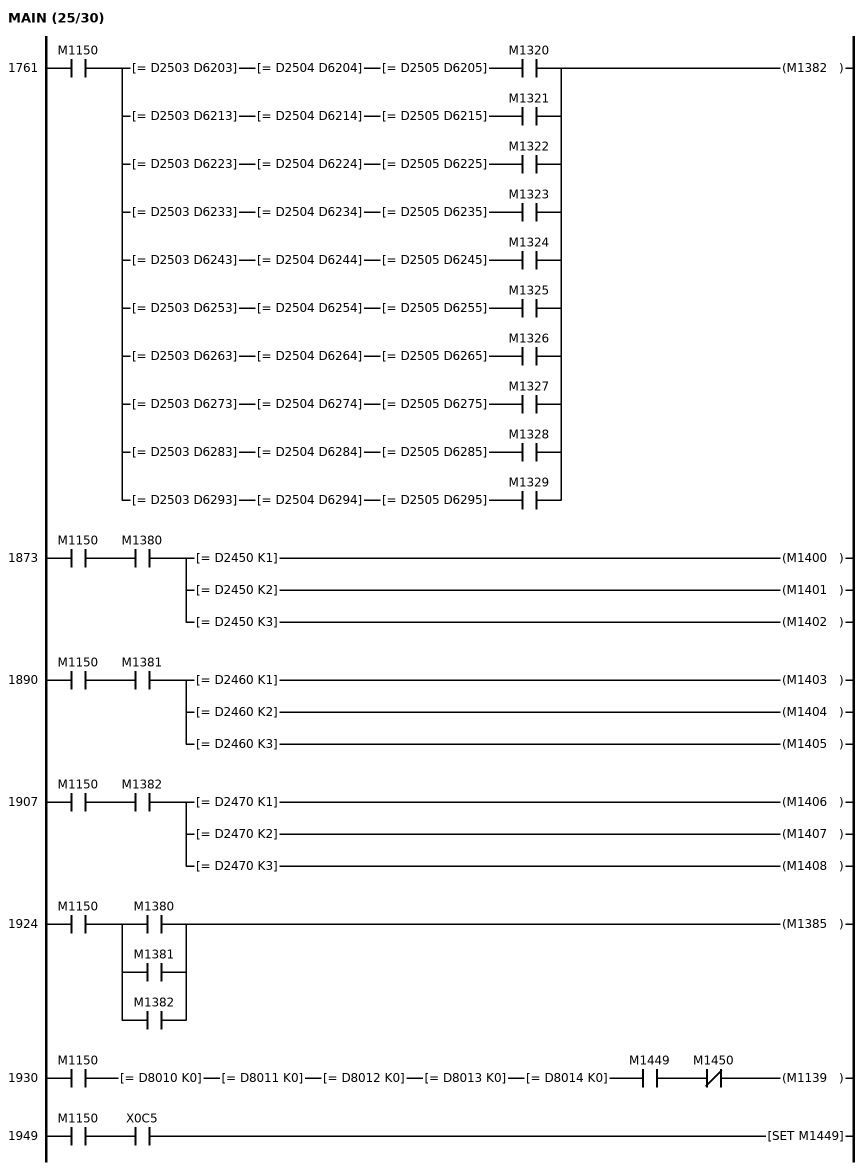
[picture p24: ladder of MAIN, rungs at steps 1761 to 1949]
1761  LD      M1150
      LD=     D2503 D6203
      AND=    D2504 D6204
      AND=    D2505 D6205
      AND     M1320
      LD=     D2503 D6213
      AND=    D2504 D6214
      AND=    D2505 D6215
      AND     M1321
      ORB
      LD=     D2503 D6223
      AND=    D2504 D6224
      AND=    D2505 D6225
      AND     M1322
      ORB
      LD=     D2503 D6233
      AND=    D2504 D6234
      AND=    D2505 D6235
      AND     M1323
      ORB
      LD=     D2503 D6243
      AND=    D2504 D6244
      AND=    D2505 D6245
      AND     M1324
      ORB
      LD=     D2503 D6253
      AND=    D2504 D6254
      AND=    D2505 D6255
      AND     M1325
      ORB
      LD=     D2503 D6263
      AND=    D2504 D6264
      AND=    D2505 D6265
      AND     M1326
      ORB
      LD=     D2503 D6273
      AND=    D2504 D6274
      AND=    D2505 D6275
      AND     M1327
      ORB
      LD=     D2503 D6283
      AND=    D2504 D6284
      AND=    D2505 D6285
      AND     M1328
      ORB
      LD=     D2503 D6293
      AND=    D2504 D6294
      AND=    D2505 D6295
      AND     M1329
      ORB
      ANB
      OUT     M1382
1873  LD      M1150
      AND     M1380
      MPS
      AND=    D2450 K1
      OUT     M1400
      MRD
      AND=    D2450 K2
      OUT     M1401
      MPP
      AND=    D2450 K3
      OUT     M1402
1890  LD      M1150
      AND     M1381
      MPS
      AND=    D2460 K1
      OUT     M1403
      MRD
      AND=    D2460 K2
      OUT     M1404
      MPP
      AND=    D2460 K3
      OUT     M1405
1907  LD      M1150
      AND     M1382
      MPS
      AND=    D2470 K1
      OUT     M1406
      MRD
      AND=    D2470 K2
      OUT     M1407
      MPP
      AND=    D2470 K3
      OUT     M1408
1924  LD      M1150
      LD      M1380
      OR      M1381
      OR      M1382
      ANB
      OUT     M1385
1930  LD      M1150
      AND=    D8010 K0
      AND=    D8011 K0
      AND=    D8012 K0
      AND=    D8013 K0
      AND=    D8014 K0
      AND     M1449
      ANI     M1450
      OUT     M1139
1949  LD      M1150
      AND     X0C5
      SET     M1449
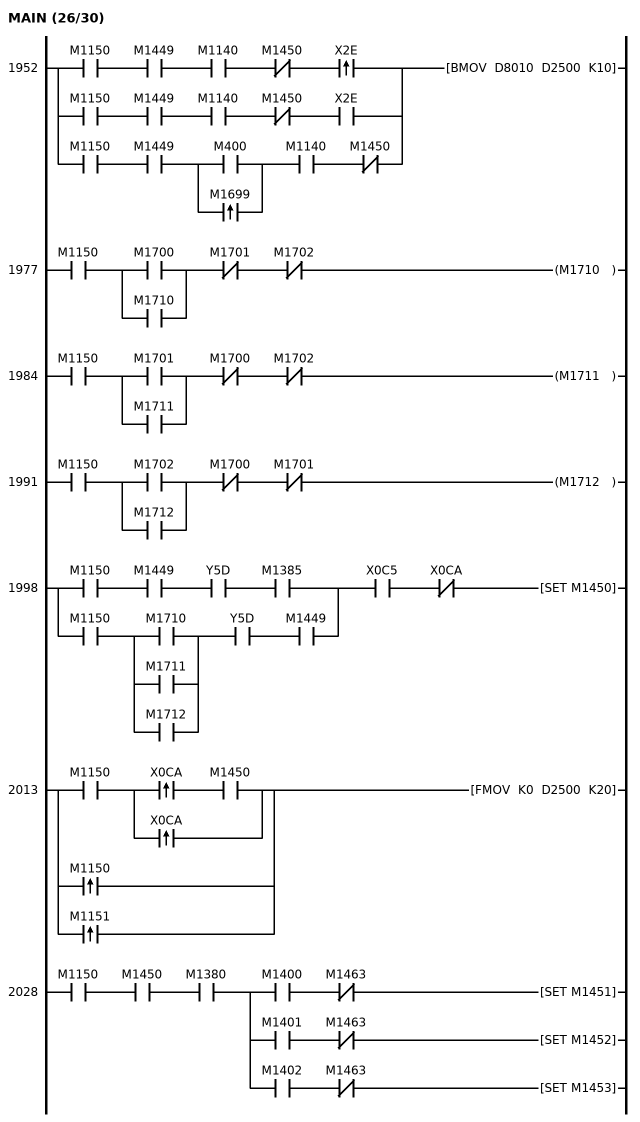
1952  LD      M1150
      AND     M1449
      AND     M1140
      ANI     M1450
      ANDP    X2E
      LD      M1150
      AND     M1449
      AND     M1140
      ANI     M1450
      AND     X2E
      ORB
      LD      M1150
      AND     M1449
      LD      M400
      ORP     M1699
      ANB
      AND     M1140
      ANI     M1450
      ORB
      BMOV    D8010 D2500 K10
1977  LD      M1150
      LD      M1700
      OR      M1710
      ANB
      ANI     M1701
      ANI     M1702
      OUT     M1710
1984  LD      M1150
      LD      M1701
      OR      M1711
      ANB
      ANI     M1700
      ANI     M1702
      OUT     M1711
1991  LD      M1150
      LD      M1702
      OR      M1712
      ANB
      ANI     M1700
      ANI     M1701
      OUT     M1712
1998  LD      M1150
      AND     M1449
      AND     Y5D
      AND     M1385
      LD      M1150
      LD      M1710
      OR      M1711
      OR      M1712
      ANB
      AND     Y5D
      AND     M1449
      ORB
      AND     X0C5
      ANI     X0CA
      SET     M1450
2013  LD      M1150
      LDP     X0CA
      AND     M1450
      ORP     X0CA
      ANB
      ORP     M1150
      ORP     M1151
      FMOV    K0 D2500 K20
2028  LD      M1150
      AND     M1450
      AND     M1380
      MPS
      AND     M1400
      ANI     M1463
      SET     M1451
      MRD
      AND     M1401
      ANI     M1463
      SET     M1452
      MPP
      AND     M1402
      ANI     M1463
      SET     M1453
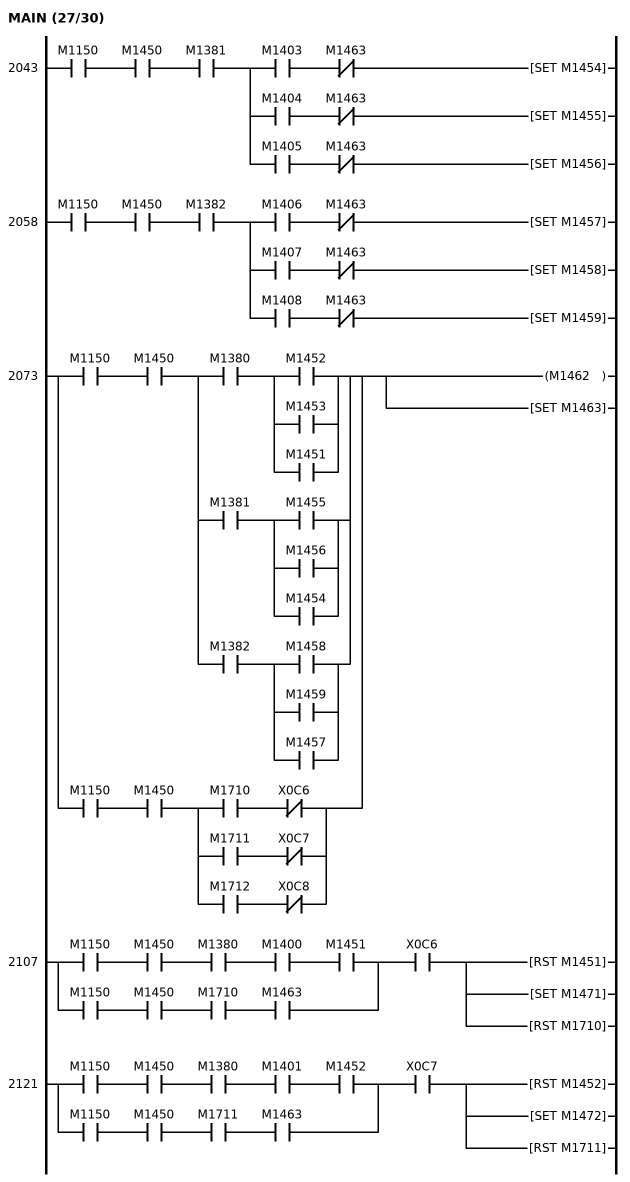
2043  LD      M1150
      AND     M1450
      AND     M1381
      MPS
      AND     M1403
      ANI     M1463
      SET     M1454
      MRD
      AND     M1404
      ANI     M1463
      SET     M1455
      MPP
      AND     M1405
      ANI     M1463
      SET     M1456
2058  LD      M1150
      AND     M1450
      AND     M1382
      MPS
      AND     M1406
      ANI     M1463
      SET     M1457
      MRD
      AND     M1407
      ANI     M1463
      SET     M1458
      MPP
      AND     M1408
      ANI     M1463
      SET     M1459
2073  LD      M1150
      AND     M1450
      LD      M1380
      LD      M1452
      OR      M1453
      OR      M1451
      ANB
      LD      M1381
      LD      M1455
      OR      M1456
      OR      M1454
      ANB
      ORB
      LD      M1382
      LD      M1458
      OR      M1459
      OR      M1457
      ANB
      ORB
      ANB
      LD      M1150
      AND     M1450
      LD      M1710
      ANI     X0C6
      LD      M1711
      ANI     X0C7
      ORB
      LD      M1712
      ANI     X0C8
      ORB
      ANB
      ORB
      OUT     M1462
      SET     M1463
2107  LD      M1150
      AND     M1450
      AND     M1380
      AND     M1400
      AND     M1451
      LD      M1150
      AND     M1450
      AND     M1710
      AND     M1463
      ORB
      AND     X0C6
      RST     M1451
      SET     M1471
      RST     M1710
2121  LD      M1150
      AND     M1450
      AND     M1380
      AND     M1401
      AND     M1452
      LD      M1150
      AND     M1450
      AND     M1711
      AND     M1463
      ORB
      AND     X0C7
      RST     M1452
      SET     M1472
      RST     M1711
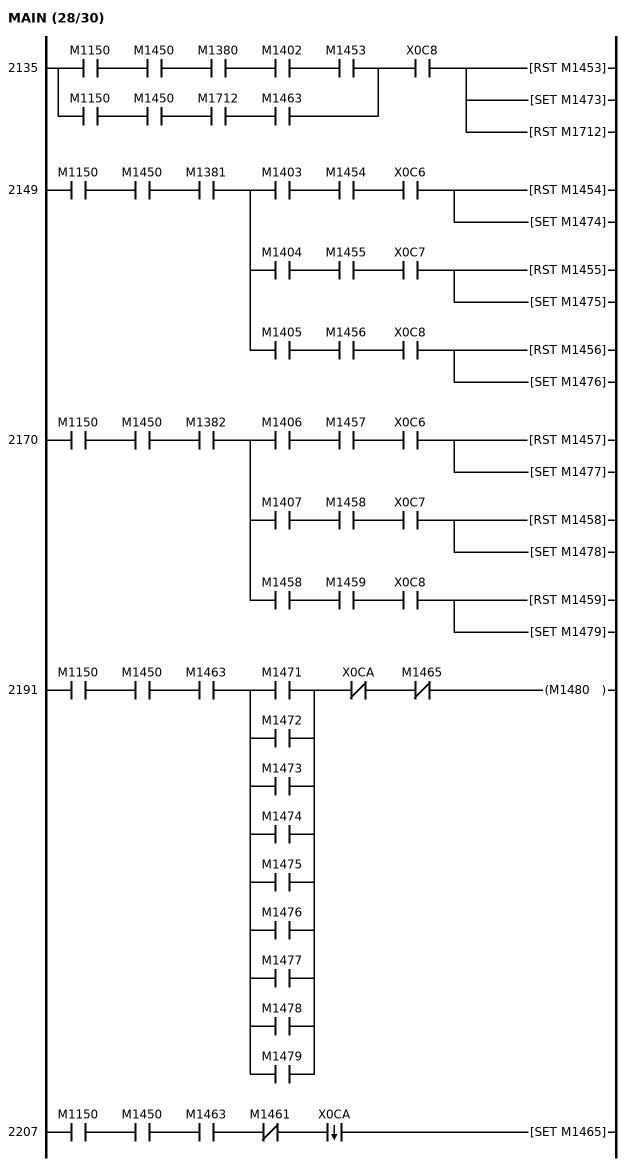
2135  LD      M1150
      AND     M1450
      AND     M1380
      AND     M1402
      AND     M1453
      LD      M1150
      AND     M1450
      AND     M1712
      AND     M1463
      ORB
      AND     X0C8
      RST     M1453
      SET     M1473
      RST     M1712
2149  LD      M1150
      AND     M1450
      AND     M1381
      MPS
      AND     M1403
      AND     M1454
      AND     X0C6
      RST     M1454
      SET     M1474
      MRD
      AND     M1404
      AND     M1455
      AND     X0C7
      RST     M1455
      SET     M1475
      MPP
      AND     M1405
      AND     M1456
      AND     X0C8
      RST     M1456
      SET     M1476
2170  LD      M1150
      AND     M1450
      AND     M1382
      MPS
      AND     M1406
      AND     M1457
      AND     X0C6
      RST     M1457
      SET     M1477
      MRD
      AND     M1407
      AND     M1458
      AND     X0C7
      RST     M1458
      SET     M1478
      MPP
      AND     M1458
      AND     M1459
      AND     X0C8
      RST     M1459
      SET     M1479
2191  LD      M1150
      AND     M1450
      AND     M1463
      LD      M1471
      OR      M1472
      OR      M1473
      OR      M1474
      OR      M1475
      OR      M1476
      OR      M1477
      OR      M1478
      OR      M1479
      ANB
      ANI     X0CA
      ANI     M1465
      OUT     M1480
2207  LD      M1150
      AND     M1450
      AND     M1463
      ANI     M1461
      ANDF    X0CA
      SET     M1465
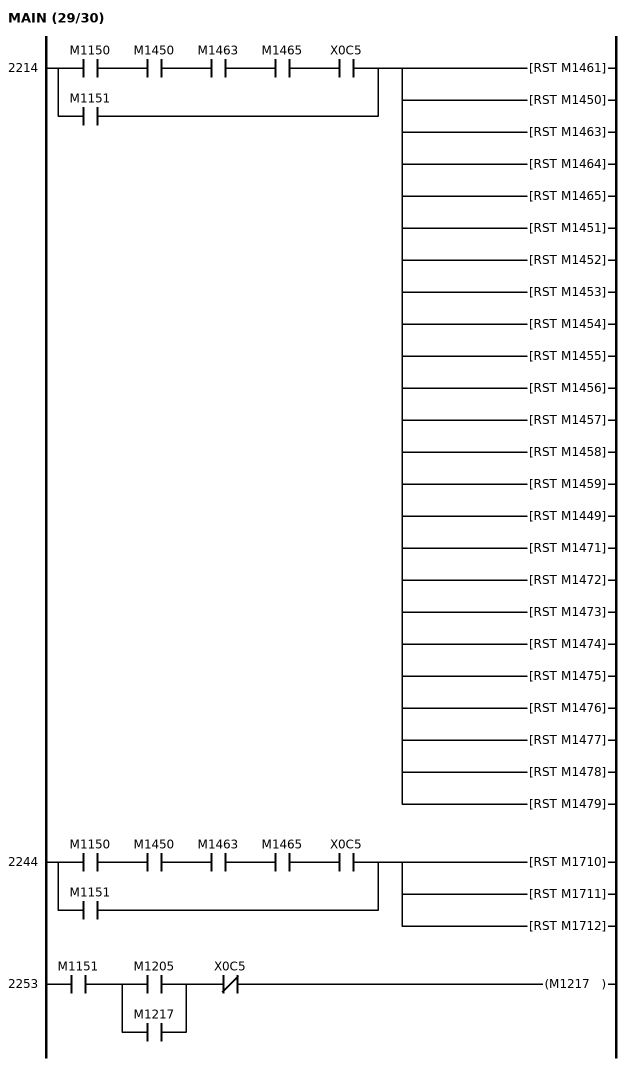
2214  LD      M1150
      AND     M1450
      AND     M1463
      AND     M1465
      AND     X0C5
      OR      M1151
      RST     M1461
      RST     M1450
      RST     M1463
      RST     M1464
      RST     M1465
      RST     M1451
      RST     M1452
      RST     M1453
      RST     M1454
      RST     M1455
      RST     M1456
      RST     M1457
      RST     M1458
      RST     M1459
      RST     M1449
      RST     M1471
      RST     M1472
      RST     M1473
      RST     M1474
      RST     M1475
      RST     M1476
      RST     M1477
      RST     M1478
      RST     M1479
2244  LD      M1150
      AND     M1450
      AND     M1463
      AND     M1465
      AND     X0C5
      OR      M1151
      RST     M1710
      RST     M1711
      RST     M1712
2253  LD      M1151
      LD      M1205
      OR      M1217
      ANB
      ANI     X0C5
      OUT     M1217
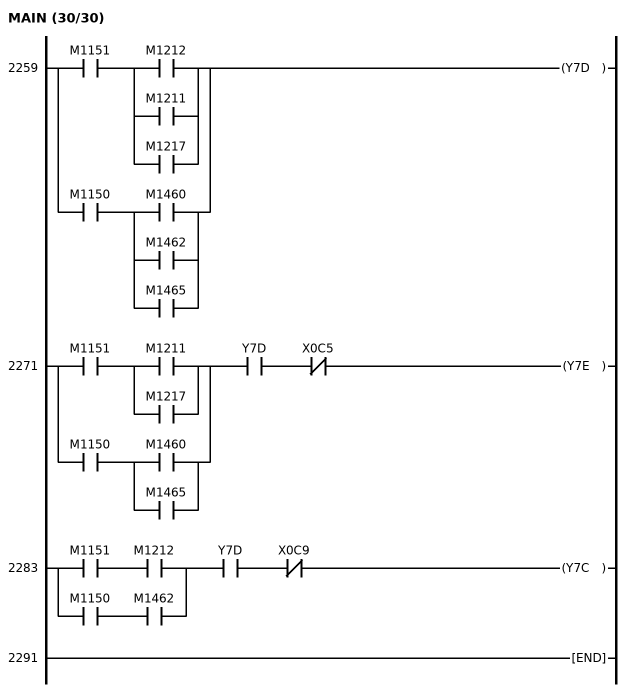
2259  LD      M1151
      LD      M1212
      OR      M1211
      OR      M1217
      ANB
      LD      M1150
      LD      M1460
      OR      M1462
      OR      M1465
      ANB
      ORB
      OUT     Y7D
2271  LD      M1151
      LD      M1211
      OR      M1217
      ANB
      LD      M1150
      LD      M1460
      OR      M1465
      ANB
      ORB
      AND     Y7D
      ANI     X0C5
      OUT     Y7E
2283  LD      M1151
      AND     M1212
      LD      M1150
      AND     M1462
      ORB
      AND     Y7D
      ANI     X0C9
      OUT     Y7C
2291  END
END_PROGRAM

PROGRAM TT_ANDON
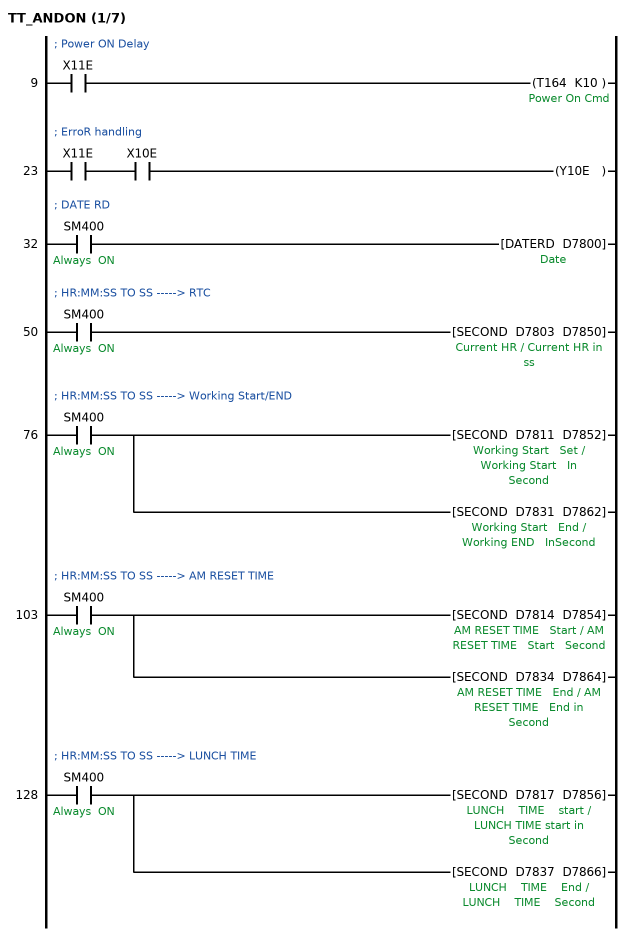
; Power ON Delay
9     LD      X11E
      OUT     T164 K10  ; Power On Cmd
; ErroR handling
23    LD      X11E
      AND     X10E
      OUT     Y10E
; DATE RD
32    LD      SM400  ; Always  ON
      DATERD  D7800  ; Date
; HR:MM:SS TO SS -----> RTC
50    LD      SM400  ; Always  ON
      SECOND  D7803 D7850  ; Current HR / Current HR in ss
; HR:MM:SS TO SS -----> Working Start/END
76    LD      SM400  ; Always  ON
      SECOND  D7811 D7852  ; Working Start   Set / Working Start   In      Second
      SECOND  D7831 D7862  ; Working Start   End / Working END   InSecond
; HR:MM:SS TO SS -----> AM RESET TIME
103   LD      SM400  ; Always  ON
      SECOND  D7814 D7854  ; AM RESET TIME   Start / AM RESET TIME   Start   Second
      SECOND  D7834 D7864  ; AM RESET TIME   End / AM RESET TIME   End in  Second
; HR:MM:SS TO SS -----> LUNCH TIME
128   LD      SM400  ; Always  ON
      SECOND  D7817 D7856  ; LUNCH    TIME    start / LUNCH TIME start in     Second
      SECOND  D7837 D7866  ; LUNCH    TIME    End / LUNCH    TIME    Second
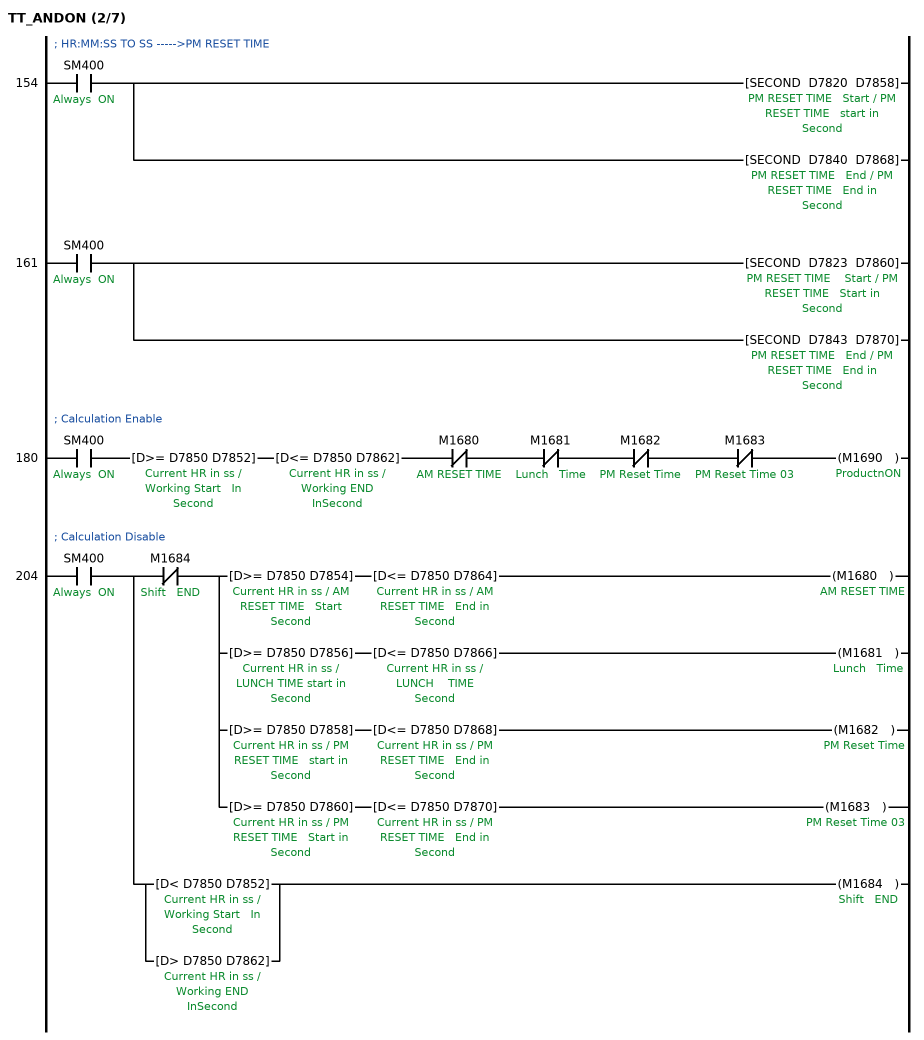
; HR:MM:SS TO SS ----->PM RESET TIME
154   LD      SM400  ; Always  ON
      SECOND  D7820 D7858  ; PM RESET TIME   Start / PM RESET TIME   start in Second
      SECOND  D7840 D7868  ; PM RESET TIME   End / PM RESET TIME   End in  Second
161   LD      SM400  ; Always  ON
      SECOND  D7823 D7860  ; PM RESET TIME    Start / PM RESET TIME   Start in Second
      SECOND  D7843 D7870  ; PM RESET TIME   End / PM RESET TIME   End in  Second
; Calculation Enable
180   LD      SM400  ; Always  ON
      ANDD>=  D7850 D7852  ; Current HR in ss / Working Start   In      Second
      ANDD<=  D7850 D7862  ; Current HR in ss / Working END   InSecond
      ANI     M1680  ; AM RESET TIME
      ANI     M1681  ; Lunch   Time
      ANI     M1682  ; PM Reset Time
      ANI     M1683  ; PM Reset Time 03
      OUT     M1690  ; ProductnON
; Calculation Disable
204   LD      SM400  ; Always  ON
      MPS
      ANI     M1684  ; Shift   END
      MPS
      ANDD>=  D7850 D7854  ; Current HR in ss / AM RESET TIME   Start   Second
      ANDD<=  D7850 D7864  ; Current HR in ss / AM RESET TIME   End in  Second
      OUT     M1680  ; AM RESET TIME
      MRD
      ANDD>=  D7850 D7856  ; Current HR in ss / LUNCH TIME start in     Second
      ANDD<=  D7850 D7866  ; Current HR in ss / LUNCH    TIME    Second
      OUT     M1681  ; Lunch   Time
      MRD
      ANDD>=  D7850 D7858  ; Current HR in ss / PM RESET TIME   start in Second
      ANDD<=  D7850 D7868  ; Current HR in ss / PM RESET TIME   End in  Second
      OUT     M1682  ; PM Reset Time
      MPP
      ANDD>=  D7850 D7860  ; Current HR in ss / PM RESET TIME   Start in Second
      ANDD<=  D7850 D7870  ; Current HR in ss / PM RESET TIME   End in  Second
      OUT     M1683  ; PM Reset Time 03
      MPP
      LDD<    D7850 D7852  ; Current HR in ss / Working Start   In      Second
      ORD>    D7850 D7862  ; Current HR in ss / Working END   InSecond
      ANB
      OUT     M1684  ; Shift   END
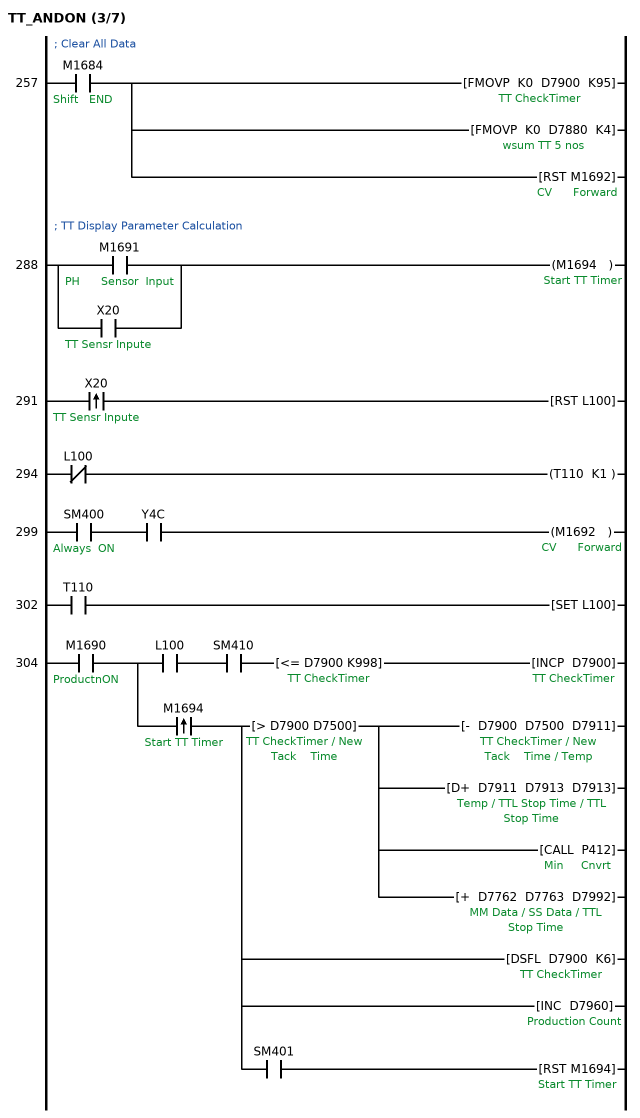
; Clear All Data
257   LD      M1684  ; Shift   END
      FMOVP   K0 D7900 K95  ; TT CheckTimer
      FMOVP   K0 D7880 K4  ; wsum TT 5 nos
      RST     M1692  ; CV      Forward
; TT Display Parameter Calculation
288   LD      M1691  ; PH      Sensor  Input
      OR      X20  ; TT Sensr Inpute
      OUT     M1694  ; Start TT Timer
291   LDP     X20  ; TT Sensr Inpute
      RST     L100
294   LDI     L100
      OUT     T110 K1
299   LD      SM400  ; Always  ON
      AND     Y4C
      OUT     M1692  ; CV      Forward
302   LD      T110
      SET     L100
304   LD      M1690  ; ProductnON
      MPS
      AND     L100
      AND     SM410
      AND<=   D7900 K998  ; TT CheckTimer
      INCP    D7900
      MPP
      ANDP    M1694  ; Start TT Timer
      MPS
      AND>    D7900 D7500  ; TT CheckTimer / New     Tack    Time
      -       D7900 D7500 D7911  ; Temp
      D+      D7911 D7913 D7913  ; TTL Stop Time
      CALL    P412  ; Min     Cnvrt
      +       D7762 D7763 D7992  ; MM Data / SS Data / TTL Stop Time
      MPP
      DSFL    D7900 K6
      INC     D7960  ; Production Count
      AND     SM401
      RST     M1694  ; Start TT Timer
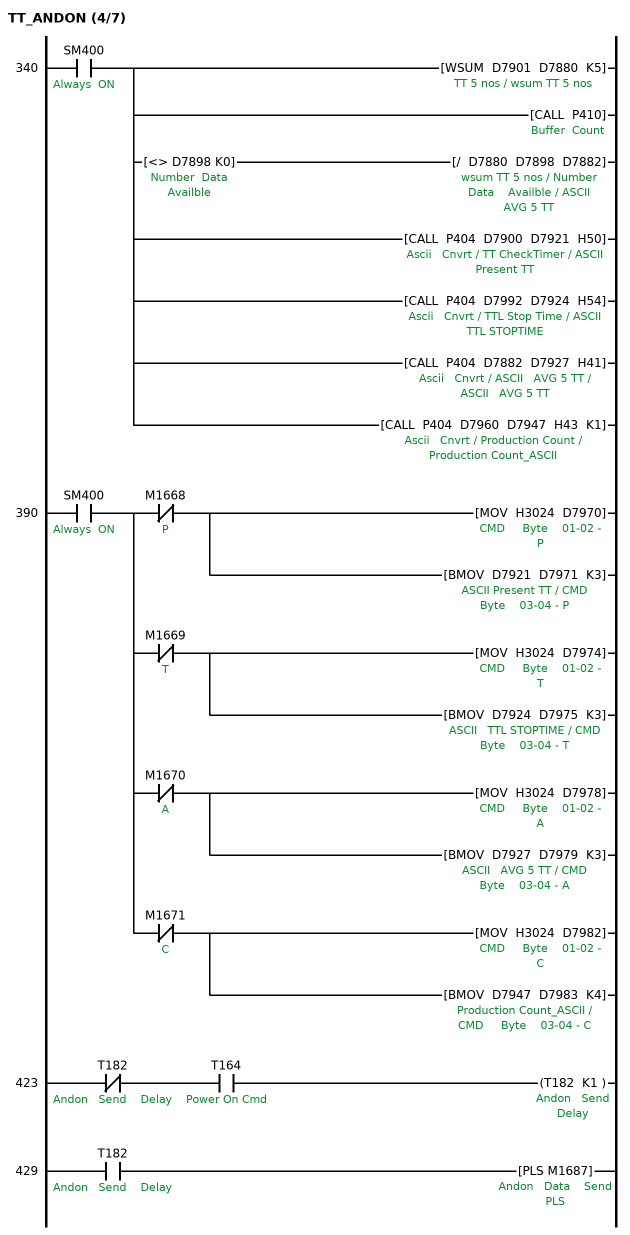
340   LD      SM400  ; Always  ON
      WSUM    D7901 D7880 K5  ; TT 5 nos
      CALL    P410  ; Buffer  Count
      MPS
      AND<>   D7898 K0  ; Number  Data    Availble
      /       D7880 D7898 D7882  ; ASCII   AVG 5 TT
        [note] 
      MPP
      CALL    P404 D7900 D7921 H50  ; Ascii   Cnvrt / ASCII Present TT
        [note] 
      CALL    P404 D7992 D7924 H54  ; ASCII   TTL STOPTIME
        [note] 
      CALL    P404 D7882 D7927 H41  ; ASCII   AVG 5 TT
        [note] 
      CALL    P404 D7960 D7947 H43 K1  ; Production Count_ASCII
        [note] 43 : C : Command
390   LD      SM400  ; Always  ON
      MPS
      ANI     M1668  ; P
      MOV     H3024 D7970  ; CMD     Byte    01-02 - P
      BMOV    D7921 D7971 K3  ; CMD     Byte    03-04 - P
      MRD
      ANI     M1669  ; T
      MOV     H3024 D7974  ; CMD     Byte    01-02 - T
      BMOV    D7924 D7975 K3  ; CMD     Byte    03-04 - T
      MRD
      ANI     M1670  ; A
      MOV     H3024 D7978  ; CMD     Byte    01-02 - A
      BMOV    D7927 D7979 K3  ; CMD     Byte    03-04 - A
      MPP
      ANI     M1671  ; C
      MOV     H3024 D7982  ; CMD     Byte    01-02 - C
      BMOV    D7947 D7983 K4  ; CMD     Byte    03-04 - C
423   LDI     T182  ; Andon   Send    Delay
      AND     T164  ; Power On Cmd
      OUT     T182 K1  ; Andon   Send    Delay
429   LD      T182  ; Andon   Send    Delay
      PLS     M1687  ; Andon   Data    Send PLS
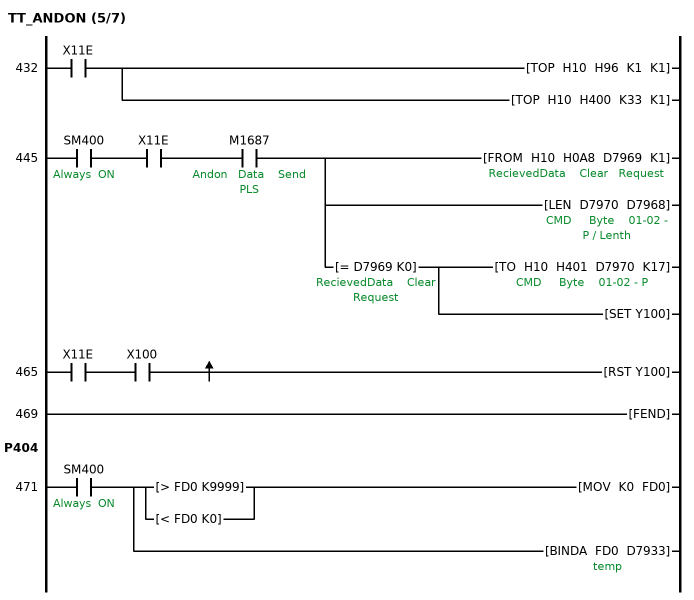
432   LD      X11E
      TOP     H10 H96 K1 K1
      TOP     H10 H400 K33 K1
445   LD      SM400  ; Always  ON
      AND     X11E
      AND     M1687  ; Andon   Data    Send PLS
      FROM    H10 H0A8 D7969 K1  ; RecievedData    Clear   Request
      LEN     D7970 D7968  ; Lenth
      AND=    D7969 K0  ; RecievedData    Clear   Request
      TO      H10 H401 D7970 K17
      SET     Y100
465   LD      X11E
      AND     X100
      MEP
      RST     Y100
469   FEND
      P404
471   LD      SM400  ; Always  ON
      MPS
      LD>     FD0 K9999
      OR<     FD0 K0
      ANB
      MOV     K0 FD0
      MPP
      BINDA   FD0 D7933  ; temp
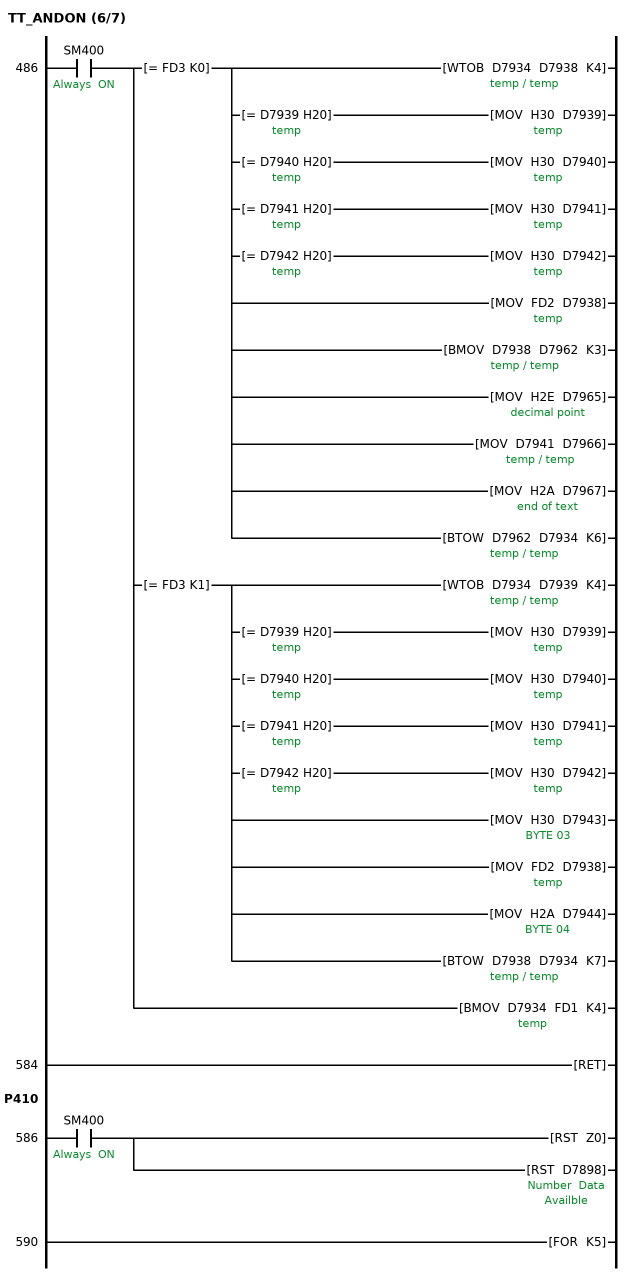
486   LD      SM400  ; Always  ON
      MPS
      AND=    FD3 K0
      WTOB    D7934 D7938 K4  ; temp / temp
      MPS
      AND=    D7939 H20  ; temp
      MOV     H30 D7939
      MRD
      AND=    D7940 H20  ; temp
      MOV     H30 D7940
      MRD
      AND=    D7941 H20  ; temp
      MOV     H30 D7941
      MRD
      AND=    D7942 H20  ; temp
      MOV     H30 D7942
      MPP
      MOV     FD2 D7938
      BMOV    D7938 D7962 K3  ; temp
      MOV     H2E D7965  ; decimal point
      MOV     D7941 D7966  ; temp
      MOV     H2A D7967  ; end of text
      BTOW    D7962 D7934 K6
      MRD
      AND=    FD3 K1
      WTOB    D7934 D7939 K4
      MPS
      AND=    D7939 H20  ; temp
      MOV     H30 D7939
      MRD
      AND=    D7940 H20  ; temp
      MOV     H30 D7940
      MRD
      AND=    D7941 H20  ; temp
      MOV     H30 D7941
      MRD
      AND=    D7942 H20  ; temp
      MOV     H30 D7942
      MPP
      MOV     H30 D7943  ; BYTE 03
      MOV     FD2 D7938
      MOV     H2A D7944  ; BYTE 04
      BTOW    D7938 D7934 K7
      MPP
      BMOV    D7934 FD1 K4
584   RET
      P410
586   LD      SM400  ; Always  ON
      RST     Z0
      RST     D7898  ; Number  Data    Availble
590   FOR     K5
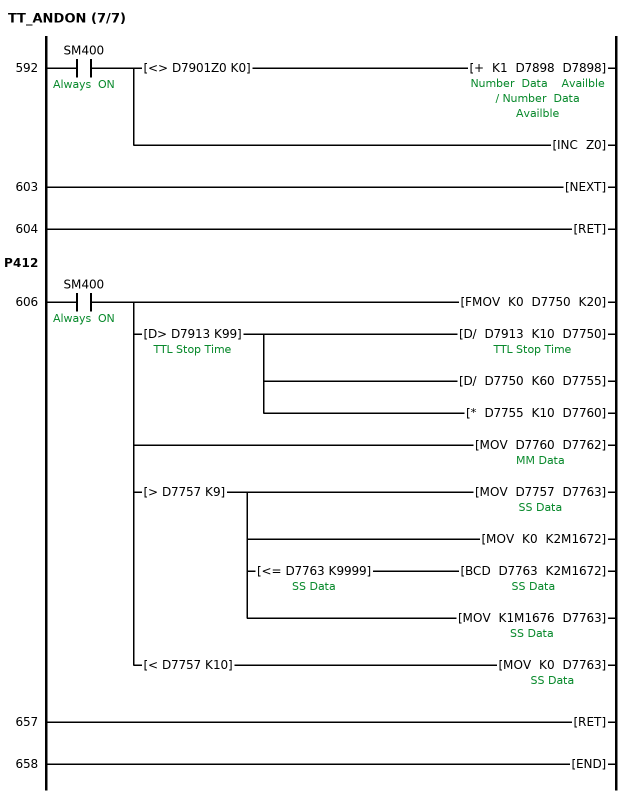
592   LD      SM400  ; Always  ON
      MPS
      AND<>   D7901Z0 K0
      +       K1 D7898 D7898
      MPP
      INC     Z0
603   NEXT
604   RET
      P412
606   LD      SM400  ; Always  ON
      FMOV    K0 D7750 K20
      MPS
      ANDD>   D7913 K99  ; TTL Stop Time
      D/      D7913 K10 D7750
      D/      D7750 K60 D7755
      *       D7755 K10 D7760
      MPP
      MOV     D7760 D7762
      MPS
      AND>    D7757 K9
      MOV     D7757 D7763
      MOV     K0 K2M1672
      MPS
      AND<=   D7763 K9999  ; SS Data
      BCD     D7763 K2M1672
      MPP
      MOV     K1M1676 D7763
      MPP
      AND<    D7757 K10
      MOV     K0 D7763
657   RET
658   END
END_PROGRAM

// device comments not shown above
D7892  ; ASCII   TTL STOPTIME
D7950  ; Sum of  TT 5 Nos
D7952  ; AVG 5 TT
L1000  ; Force
